FUNCTION_BLOCK GreenMasterXXL EXTENDS GreenMasterBase
VAR PERSISTENT
	ParametersXXL: GreenMasterParametersXXL;
END_VAR
VAR_INPUT
END_VAR
VAR_OUTPUT
END_VAR
VAR
	SupplyFanControl: FanControl;
	ExtractFanControl: FanControl;
	Recirculation: BOOL;
	VentilationControl: VentilationControl;
	ExhaustAir: BOOL;
	SupplyAir: BOOL := TRUE;
	StopVentilation: bool;

	ExtractFanPV: LREAL;
	SupplyFanPV: LREAL;
	Defrost_0: Defrost;
	WriteLRealIf_0: WriteLRealIf;
END_VAR
VAR // added by the converter: edge detectors and wires of the graphical bodies
    _w1, _w2, _w3, _w4, _w5, _w6 : ANY;
END_VAR


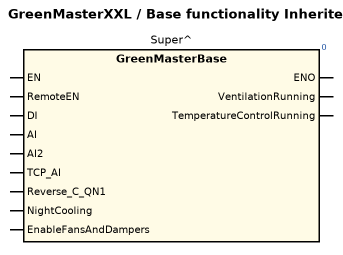
// PAGE Base functionality Inherited from greenMasterBase
Super^(); // GreenMasterBase

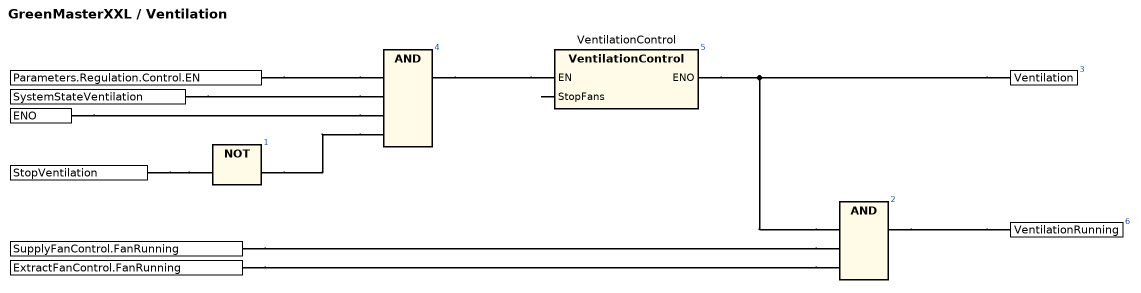
// PAGE Ventilation
_w1 := VentilationControl.ENO AND SupplyFanControl.FanRunning AND ExtractFanControl.FanRunning;
Ventilation := VentilationControl.ENO;
VentilationControl(EN := Parameters.Regulation.Control.EN AND SystemStateVentilation AND ENO AND NOT StopVentilation);
VentilationRunning := _w1;

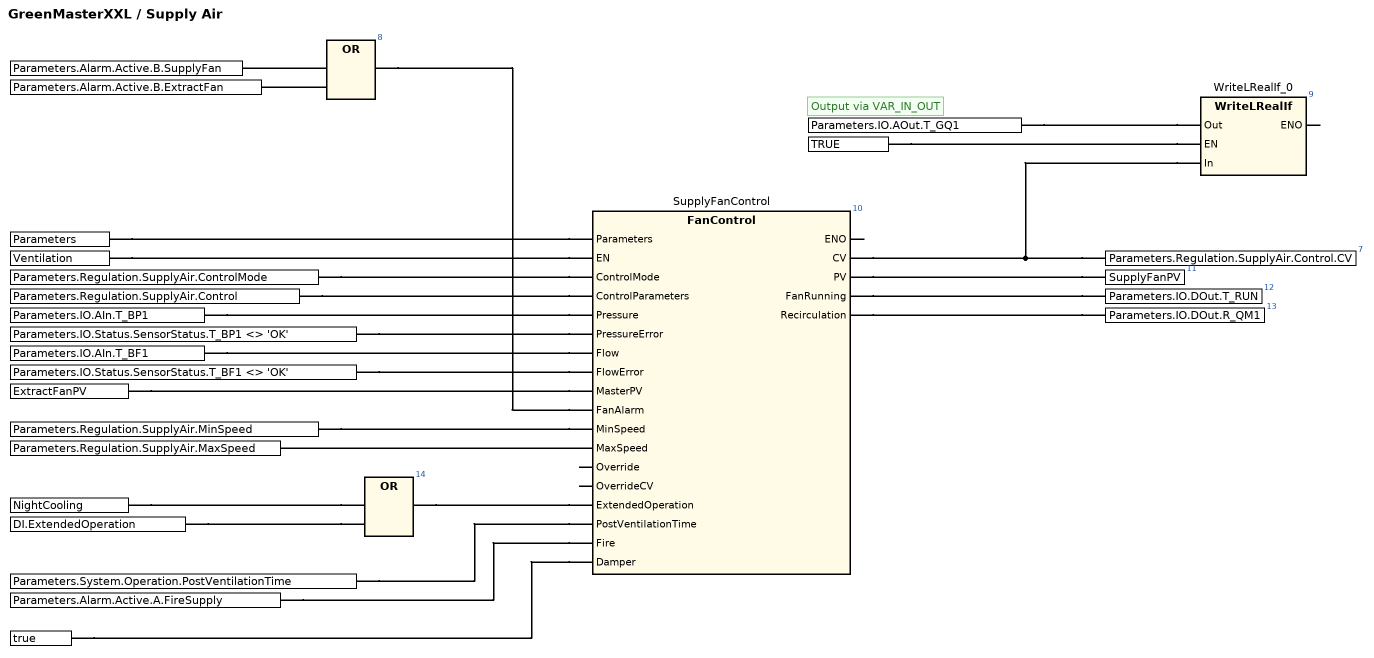
// PAGE Supply Air
Parameters.Regulation.SupplyAir.Control.CV := SupplyFanControl.CV;
_w2 := Parameters.Alarm.Active.B.SupplyFan OR Parameters.Alarm.Active.B.ExtractFan;
WriteLRealIf_0(Out := Parameters.IO.AOut.T_GQ1, EN := TRUE, In := SupplyFanControl.CV); // WriteLRealIf
// Output via VAR_IN_OUT
SupplyFanControl(
    Parameters := Parameters,
    EN := Ventilation,
    ControlMode := Parameters.Regulation.SupplyAir.ControlMode,
    ControlParameters := Parameters.Regulation.SupplyAir.Control,
    Pressure := Parameters.IO.AIn.T_BP1,
    PressureError := Parameters.IO.Status.SensorStatus.T_BP1 <> 'OK',
    Flow := Parameters.IO.AIn.T_BF1,
    FlowError := Parameters.IO.Status.SensorStatus.T_BF1 <> 'OK',
    MasterPV := ExtractFanPV,
    FanAlarm := _w2,
    MinSpeed := Parameters.Regulation.SupplyAir.MinSpeed,
    MaxSpeed := Parameters.Regulation.SupplyAir.MaxSpeed,
    ExtendedOperation := _w3,
    PostVentilationTime := Parameters.System.Operation.PostVentilationTime,
    Fire := Parameters.Alarm.Active.A.FireSupply,
    Damper := true); // FanControl
SupplyFanPV := SupplyFanControl.PV;
Parameters.IO.DOut.T_RUN := SupplyFanControl.FanRunning;
Parameters.IO.DOut.R_QM1 := SupplyFanControl.Recirculation;
_w3 := NightCooling OR DI.ExtendedOperation;

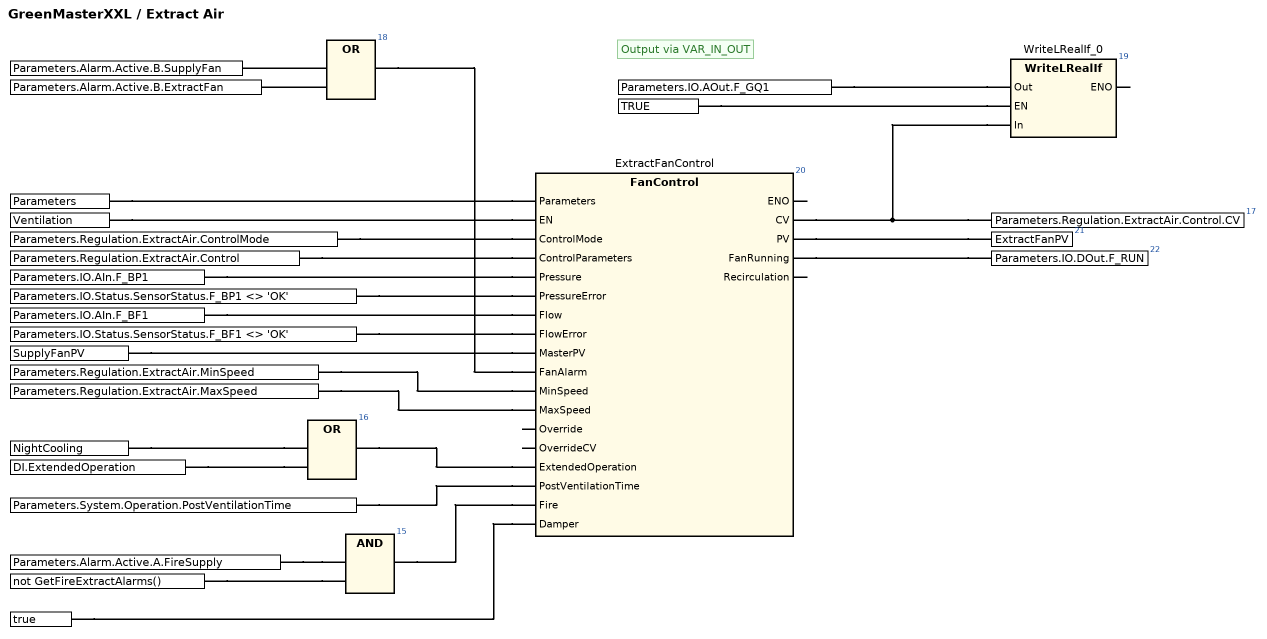
// PAGE Extract Air
_w4 := Parameters.Alarm.Active.A.FireSupply AND (not GetFireExtractAlarms());
_w5 := NightCooling OR DI.ExtendedOperation;
Parameters.Regulation.ExtractAir.Control.CV := ExtractFanControl.CV;
_w6 := Parameters.Alarm.Active.B.SupplyFan OR Parameters.Alarm.Active.B.ExtractFan;
WriteLRealIf_0(Out := Parameters.IO.AOut.F_GQ1, EN := TRUE, In := ExtractFanControl.CV); // WriteLRealIf
// Output via VAR_IN_OUT
ExtractFanControl(
    Parameters := Parameters,
    EN := Ventilation,
    ControlMode := Parameters.Regulation.ExtractAir.ControlMode,
    ControlParameters := Parameters.Regulation.ExtractAir.Control,
    Pressure := Parameters.IO.AIn.F_BP1,
    PressureError := Parameters.IO.Status.SensorStatus.F_BP1 <> 'OK',
    Flow := Parameters.IO.AIn.F_BF1,
    FlowError := Parameters.IO.Status.SensorStatus.F_BF1 <> 'OK',
    MasterPV := SupplyFanPV,
    FanAlarm := _w6,
    MinSpeed := Parameters.Regulation.ExtractAir.MinSpeed,
    MaxSpeed := Parameters.Regulation.ExtractAir.MaxSpeed,
    ExtendedOperation := _w5,
    PostVentilationTime := Parameters.System.Operation.PostVentilationTime,
    Fire := _w4,
    Damper := true); // FanControl
ExtractFanPV := ExtractFanControl.PV;
Parameters.IO.DOut.F_RUN := ExtractFanControl.FanRunning;

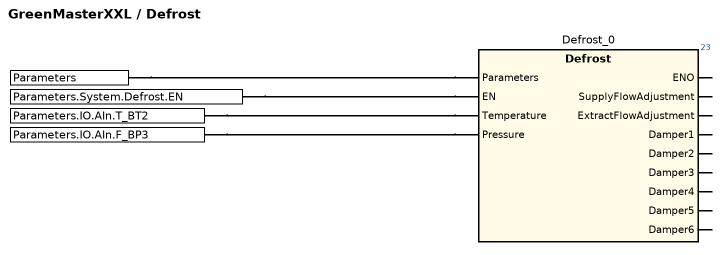
// PAGE Defrost
Defrost_0(
    Parameters := Parameters,
    EN := Parameters.System.Defrost.EN,
    Temperature := Parameters.IO.AIn.T_BT2,
    Pressure := Parameters.IO.AIn.F_BP3); // Defrost

METHOD ExtractFanOverride : BOOL
VAR_INPUT
	Override: BOOL;
	Speed: LREAL;
END_VAR
ExtractFanControl.Override := Override;
ExtractFanControl.OverrideCV := Speed;
END_METHOD

METHOD Fire : BOOL
VAR_INPUT
END_VAR
SUPER^.Fire();
SupplyFanControl.Override := Parameters.Regulation.SupplyAir.Fire.EN;
SupplyFanControl.OverrideCV := Parameters.Regulation.SupplyAir.Fire.Speed;
ExtractFanControl.Override := Parameters.Regulation.ExtractAir.Fire.EN;
ExtractFanControl.OverrideCV := Parameters.Regulation.ExtractAir.Fire.Speed;
END_METHOD

METHOD FireEnd : BOOL
VAR_INPUT
END_VAR
SUPER^.FireEnd();
SupplyFanControl.Override := FALSE;
SupplyFanControl.OverrideCV := 0;
ExtractFanControl.Override := FALSE;
ExtractFanControl.OverrideCV := 0;
END_METHOD

METHOD FireSupply : BOOL
VAR_INPUT
END_VAR
SUPER^.FireSupply();
CloseDampers();
StopVentilation := TRUE;
END_METHOD

METHOD FireSupplyEnd : BOOL
VAR_INPUT
END_VAR
SUPER^.FireSupplyEnd();
StopVentilation := FALSE;
END_METHOD

METHOD GetParametersXXL : REFERENCE TO GreenMasterParametersXXL
VAR_INPUT
END_VAR
GetParametersXXL := ParametersXXL;
END_METHOD

METHOD SetFullHeatRecovery : BOOL
VAR_INPUT
END_VAR
OvrTemperatureControl := TRUE;
OvrTemperatureCV := 0.75;
END_METHOD

{attribute 'TcRpcEnable'}
METHOD Sum : LREAL
VAR_INPUT
	v1: LREAL;
	v2: LREAL;
END_VAR
Sum := v1 + v2;
END_METHOD

METHOD SupplyFanOverride : BOOL
VAR_INPUT
	Override: BOOL;
	Speed: LREAL;
END_VAR
SupplyFanControl.Override := Override;
SupplyFanControl.OverrideCV := Speed;
END_METHOD

METHOD Update : BOOL
VAR_INPUT
	DO_: REFERENCE TO GreenMasterDO_Base;
	AO: REFERENCE TO GreenMasterAO_Base;
END_VAR
SUPER^.Update(DO_, AO);
IF Parameters.System.Operation.EN THEN
	SupplyAir := NOT Recirculation;	
END_IF
END_METHOD

END_FUNCTION_BLOCK

(* stored: Version 1.1.0.1, ProductVersion 3.1.4024.6
   POU GreenMasterXXL: Id {5f0cde82-8a2d-4f75-8383-693037e98205}, SpecialFunc None
   Method ExtractFanOverride: Id {845c6049-375f-4348-bb58-2001bb90466c}
   Method Fire: Id {1c88f70e-4e58-403a-8538-cb81e4801757}
   Method FireEnd: Id {655f18e4-a158-4a17-b2b0-9ab9f6f78de3}
   Method FireSupply: Id {307b7e85-67b1-428f-a760-6fc8536c3bc8}
   Method FireSupplyEnd: Id {b5288274-2e3c-4bbf-9853-2b400a0b0f4f}
   Method GetParametersXXL: Id {993c232f-881e-4f3c-a515-bd8ca9119aaf}
   Method SetFullHeatRecovery: Id {dfea4f11-b799-4de8-a0e3-cf18887e647e}
   Method Sum: Id {a119003f-62c1-4ad0-b714-6e4d60c5e351}
   Method SupplyFanOverride: Id {8aa461d5-b7d4-4117-ba9d-e3e15222c794}
   Method Update: Id {964d34a0-56a5-4eba-b576-6bb134f2e0c5} *)
